TYPE ST_ORCA_BrandInfo :
STRUCT

	BatchID 			: STRING(255);
	GTIN 			: STRING(255);
	SKU 				: STRING(255);
	ProductionOrder 	: STRING(255);

END_STRUCT
END_TYPE

(* stored: Version 1.1.0.1, ProductVersion 3.1.4024.15
   DUT ST_ORCA_BrandInfo: Id {637935ce-dde4-47e6-acf3-4e98c57fd274} *)
